// SIMATIC S7-200 SMART project (STEP 7-Micro/WIN SMART), CPU SR40

SYMBOL_TABLE 表格 1
过程变量             VW0
PID输出            VW2
手动输入             VD4
设定值              VD8
YLAST1           VD100
YLAST2           VD104
YLAST3           VD108
END_SYMBOL_TABLE

SYMBOL_TABLE 系统符号
Always_On        SM0.0    // 始终接通
First_Scan_On    SM0.1    // 仅在第一个扫描周期时接通
Time_1_Intrvl    SMB35    // 指定中断 1 的时间间隔（从 5 到 255，以 1 毫秒递增）。
END_SYMBOL_TABLE

ORGANIZATION_BLOCK MAIN:OB1
TITLE=程序注释
BEGIN
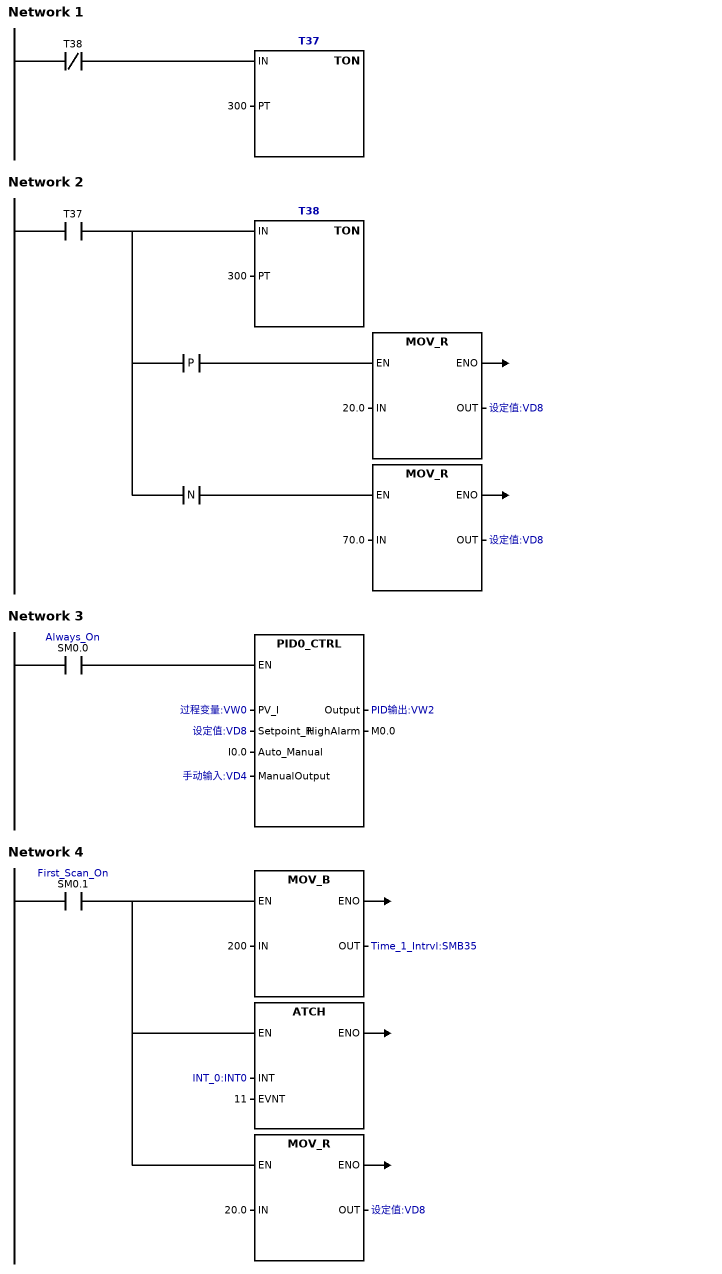
Network 1
LDN    T38
TON    T37, 300
Network 2
LD     T37
LPS
TON    T38, 300
EU
MOVR   20.0, 设定值:VD8
LPP
ED
MOVR   70.0, 设定值:VD8
Network 3
LD     Always_On:SM0.0
CALL   PID0_CTRL:SBR1, 过程变量:VW0, 设定值:VD8, I0.0, 手动输入:VD4, PID输出:VW2, M0.0
Network 4
LD     First_Scan_On:SM0.1
MOVB   200, Time_1_Intrvl:SMB35
ATCH   INT_0:INT0, 11
MOVR   20.0, 设定值:VD8
END_ORGANIZATION_BLOCK

// SBR0: protected block, not included

// SBR1: protected block, not included

INTERRUPT_BLOCK INT_0:INT0
TITLE=中断例程注释
BEGIN
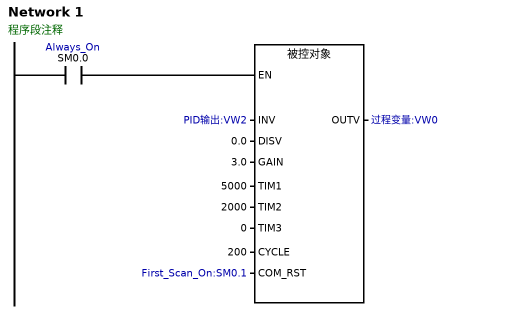
Network 1
// 程序段注释
// (network saved uncompiled; LAD cells follow)
// row 0: c0 -| |- Always_On:SM0.0  c1 --  c2 [被控对象 EN:=power@row0, INV:=PID输出:VW2, DISV:=0.0, GAIN:=3.0, TIM1:=5000, TIM2:=2000, TIM3:=0, CYCLE:=200, COM_RST:=First_Scan_On:SM0.1, OUTV=>过程变量:VW0]
// row 1: c2 [box]
// row 2: c2 [box]
// row 3: c2 [box]
END_INTERRUPT_BLOCK

// INT1: protected block, not included
